FUNCTION_BLOCK FB_SampleA_Test
VAR_INPUT
	{attribute 'pytmc' := '
		pv: fInput
		io: io
	'}
	fInput : LREAL;
END_VAR
VAR_OUTPUT
	{attribute 'pytmc' := '
		pv: fOutput
		io: input
	'}
	fOutput : LREAL;
END_VAR
VAR
END_VAR

fOutput := fInput;

END_FUNCTION_BLOCK

(* stored: Version 1.1.0.1, ProductVersion 3.1.4022.18
   POU FB_SampleA_Test: Id {5eaf07ca-8428-4095-8bca-c1835b3c56ef}, SpecialFunc None *)
